DEVICE_TYPE RMT_FRAME (* Remotely Managed Window *)
  (* Standard: 61499 ITA; Description: Remotely Managed Window *)
  (* Version 0.2, 2001-11-25, JHC, Rockwell Automation, Corrected BOUNDS comment. *)
  (* Version 0.1, 2001-08-14, JHC, Rockwell Automation, Added BOUNDS, GRID parameters. *)
  (* Version 0.0, 2001-07-26, JHC, Rockwell Automation, Replaces RMT_DEV_HMI *)
  (* Compiler header: package fb.rt.ita; import fb.rt.hmi.*; *)
  (* Compiler classdef: public class RMT_DEV_HMI extends FRAME_DEVICE implements RemoteDevice *)
  (* Compiler Java IBM VisualAge 3.0 *)
  VAR_INPUT
    BOUNDS : ARRAY [0..3] OF DINT; (* Initial[x,y,width,height] *)
    GRID : ARRAY [0..1] OF DINT; (* Grid layout[rows,cols] *)
    MGR_ID : WSTRING := "localhost:61499"; (* Device manager socket ID *)
  END_VAR
  RESOURCE MGR : RMT_RES
  END_RESOURCE
  DATA_CONNECTIONS
    MGR_ID TO MGR.MGR_ID;
  END_CONNECTIONS
END_DEVICE_TYPE
